(* LS Electric XG5000 project: Study3_TON_TOF *)
(* PLC LSPLC *)
(* module base 0 slot 0: 입력 모듈:XGI-D21A (DC 24V 입력, 8점 (전류소스/싱크입력)) *)
(* module base 0 slot 1: 출력 모듈:XGQ-RY1A (릴레이 출력, 8점 (2A용, 단독 COM.)) *)

PROGRAM NewProgram (* task: 스캔 프로그램 *)
VAR
    on AT %IX0.0.2 : BOOL;
    T1 : TON;
    T2 : TOF;
    조명 : BOOL;
END_VAR
VAR
    _e1 : R_TRIG;
END_VAR

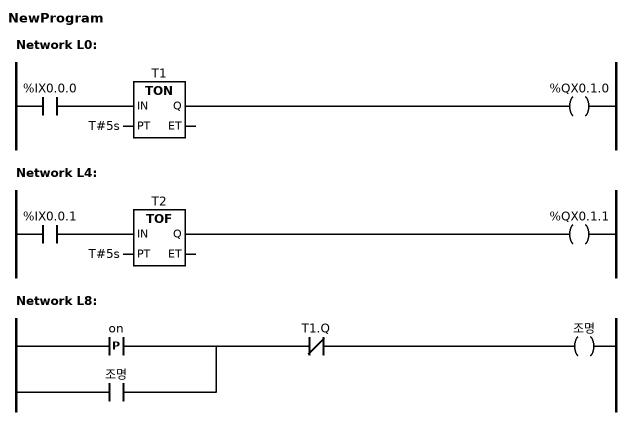
(* Rung L0 *)
T1(IN := %IX0.0.0, PT := T#5s);
%QX0.1.0 := T1.Q;
(* Rung L4 *)
T2(IN := %IX0.0.1, PT := T#5s);
%QX0.1.1 := T2.Q;
(* Rung L8 *)
_e1(CLK := on);
조명 := (_e1.Q OR 조명) AND NOT T1.Q;
END_PROGRAM